FUNCTION_BLOCK MoveMoverToPosition
VAR_INPUT
END_VAR
VAR_OUTPUT
END_VAR
VAR
	moveAbs	: MC_MoveAbsoluteCA;
	_axis : REFERENCE TO AXIS_REF;
	State: INT;
	_MoveMover : BOOL;
	_busy : BOOL;
	_error : BOOL;
	_done : BOOL;
END_VAR

CASE State OF
	0:
		IF _MoveMover THEN
			_done := FALSE;
			_error := FALSE;
			_busy := TRUE;
			moveAbs.Execute := TRUE;
			IF moveAbs.Busy THEN
				State := 10;
				_MoveMover := FALSE;
			END_IF
		END_IF
	
	10:
		IF NOT moveAbs.Busy THEN
			IF moveAbs.Done THEN
				_done := TRUE;
			ELSIF moveAbs.Error THEN
				_error := TRUE;
			END_IF
			_busy := FALSE;
			moveAbs.Execute := FALSE;
			State := 0;
		END_IF
END_CASE

moveAbs(Axis := _axis);

METHOD Abort : BOOL
moveAbs.Execute := FALSE;
moveAbs.Position := moveAbs.Velocity := 0;
_MoveMover := false;
_busy := false;
Abort := true;
State := 0;
END_METHOD

PROPERTY PUBLIC Acceleration : mc_lreal
GET
Acceleration := moveAbs.Acceleration;
END_GET
SET
moveAbs.Acceleration := Acceleration;
END_SET
END_PROPERTY

PROPERTY Busy : BOOL
GET
Busy := _busy;
END_GET
END_PROPERTY

PROPERTY PUBLIC Deceleration : mc_lreal
GET
Deceleration := moveAbs.Deceleration;
END_GET
SET
moveAbs.Deceleration := Deceleration;
END_SET
END_PROPERTY

PROPERTY Done : BOOL
GET
Done := _done;
END_GET
END_PROPERTY

PROPERTY Error : BOOL
GET
Error := _error;
END_GET
END_PROPERTY

METHOD FB_init : BOOL
VAR_INPUT
	bInitRetains : BOOL; // if TRUE, the retain variables are initialized (warm start / cold start)
	bInCopyCode : BOOL;  // if TRUE, the instance afterwards gets moved into the copy code (online change)
	axis : reference TO AXIS_REF;
END_VAR
_axis REF= axis;
END_METHOD

PROPERTY PUBLIC Gap : mc_lreal
GET
Gap := moveAbs.Gap;
END_GET
SET
moveAbs.Gap := Gap;
END_SET
END_PROPERTY

PROPERTY PUBLIC Jerk : mc_lreal
GET
Jerk := moveAbs.Jerk;
END_GET
SET
moveAbs.Jerk := Jerk;
END_SET
END_PROPERTY

METHOD MoveTo : BOOL
VAR_INPUT
	Position : MC_LREAL;
	Velocity : MC_LREAL;
END_VAR
moveAbs.Position := Position;
moveAbs.Velocity := Velocity;
_MoveMover := MoveTo := true;
END_METHOD

END_FUNCTION_BLOCK

(* stored: Version 1.1.0.1, ProductVersion 3.1.4024.6
   POU MoveMoverToPosition: Id {7bb1d5d1-744a-4af2-9a8e-f277395f1819}, SpecialFunc None
   Method Abort: Id {d5d2cfe6-b417-452e-bd46-b464683a0619}
   Property Acceleration: Id {619d3847-5c56-4d7d-8912-4a7a3c2fab53}
   Get Get: Id {160c6e4f-a16c-421d-8c0c-b9c34ac44a98}
   Set Set: Id {b31645e0-4dac-406d-9005-a1044021489d}
   Property Busy: Id {8daace01-8802-44f8-af4c-052ee1943c05}
   Get Get: Id {34dc6e2b-2d97-4490-bf69-3490dfb35bf9}
   Property Deceleration: Id {fd169959-0cda-44ca-91da-b5c02341a7b8}
   Get Get: Id {1432df43-9141-43a6-9189-a74a0b474e3a}
   Set Set: Id {9fcc36d0-7932-4cb2-99b9-ea6ac9d88e00}
   Property Done: Id {f25c1c2a-2668-4bbb-9c1e-65e8a7c684f7}
   Get Get: Id {64dd03d9-cbc3-4977-87f1-7cfb4cf220d6}
   Property Error: Id {237ec544-e3e3-45ca-b694-4a9a42a31865}
   Get Get: Id {9566cd0e-c04b-4154-896d-a3be72d0d675}
   Method FB_init: Id {c484d3f0-9bb2-42b8-9e28-4180edd6cf55}
   Property Gap: Id {bc1c3b5b-e85c-4b42-896b-71e7e3b70578}
   Get Get: Id {0acb691e-13ab-430b-be85-9e498351e353}
   Set Set: Id {6d172d01-53a2-4dc8-a168-1fce2091c957}
   Property Jerk: Id {a6c07296-6574-47b6-ba86-148f53995f4a}
   Get Get: Id {f04a9696-d447-4cb4-bf85-f8433c82c764}
   Set Set: Id {d8aeadff-43bb-4e6b-959c-377eb7731254}
   Method MoveTo: Id {5b92cfd9-e91a-4522-8c2c-ae95c78db5e8} *)
